FUNCTION_BLOCK FB_ReadCoil
VAR_INPUT
END_VAR
VAR_OUTPUT
END_VAR
VAR
END_VAR

END_FUNCTION_BLOCK

(* stored: Version 1.1.0.1, ProductVersion 3.1.4024.16
   POU FB_ReadCoil: Id {b85949c2-cea7-45da-a836-19c08f2a73fc}, SpecialFunc None *)
